Staubli VAL3: start.pgx

program start()
begin
  taskCreateSync "sender",0.5,bSender,sendData()
  taskCreateSync "receiver",0.5,bReceiver,recvData()
end
